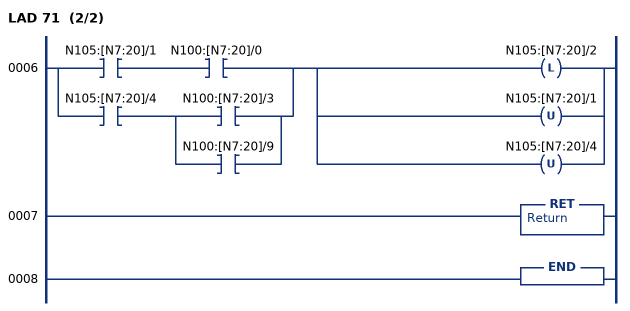
% Rung: 6 %
SOR BST XIC N105:[N7:20]/1 XIC N100:[N7:20]/0 NXB XIC N105:[N7:20]/4 BST XIC N100:[N7:20]/3 NXB XIC N100:[N7:20]/9 BND BND BST OTL N105:[N7:20]/2 NXB OTU N105:[N7:20]/1 NXB OTU N105:[N7:20]/4 BND EOR
% Rung: 7 %
SOR RET EOR
% Rung: 8 %
SOR END EOR

LADDER 75
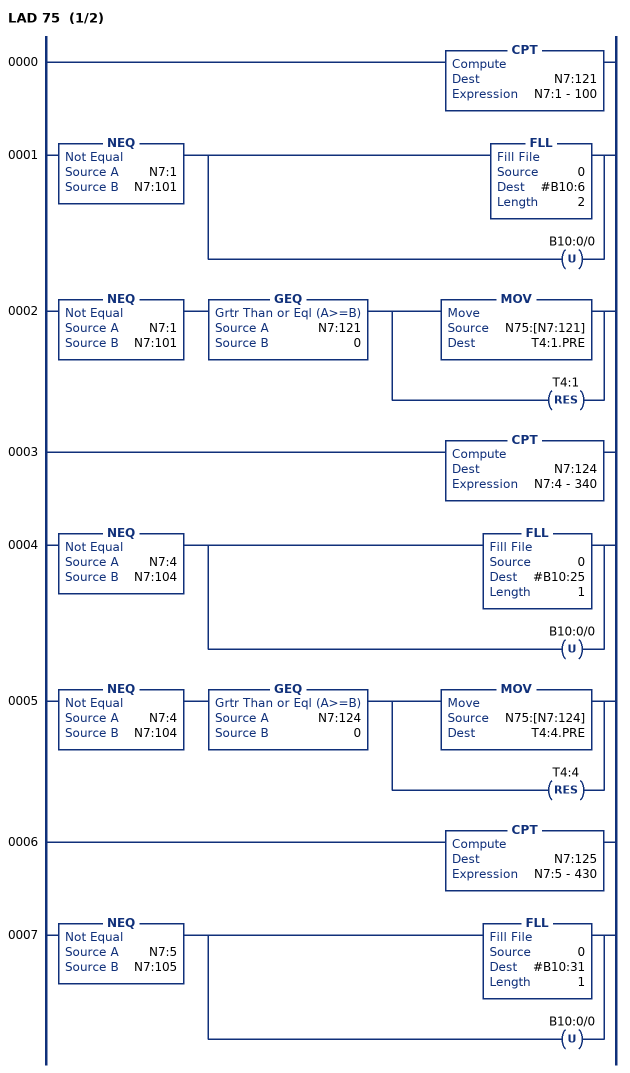
% Rung: 0 %
SOR CPT N7:121 " N7:1 - 100 " EOR
% Rung: 1 %
SOR NEQ N7:1 N7:101 BST FLL 0 #B10:6 2 NXB OTU B10:0/0 BND EOR
% Rung: 2 %
SOR NEQ N7:1 N7:101 GEQ N7:121 0 BST MOV N75:[N7:121] T4:1.PRE NXB RES T4:1 BND EOR
% Rung: 3 %
SOR CPT N7:124 " N7:4 - 340 " EOR
% Rung: 4 %
SOR NEQ N7:4 N7:104 BST FLL 0 #B10:25 1 NXB OTU B10:0/0 BND EOR
% Rung: 5 %
SOR NEQ N7:4 N7:104 GEQ N7:124 0 BST MOV N75:[N7:124] T4:4.PRE NXB RES T4:4 BND EOR
% Rung: 6 %
SOR CPT N7:125 " N7:5 - 430 " EOR
% Rung: 7 %
SOR NEQ N7:5 N7:105 BST FLL 0 #B10:31 1 NXB OTU B10:0/0 BND EOR

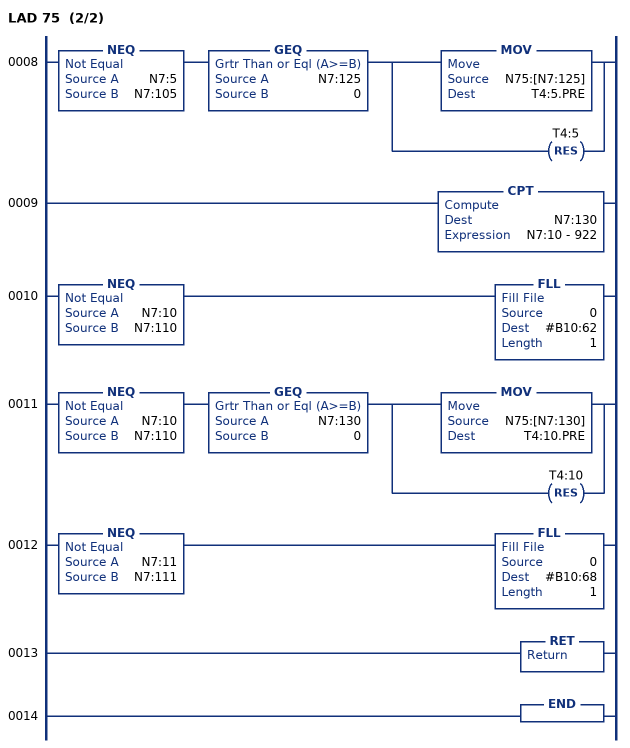
% Rung: 8 %
SOR NEQ N7:5 N7:105 GEQ N7:125 0 BST MOV N75:[N7:125] T4:5.PRE NXB RES T4:5 BND EOR
% Rung: 9 %
SOR CPT N7:130 " N7:10 - 922 " EOR
% Rung: 10 %
SOR NEQ N7:10 N7:110 FLL 0 #B10:62 1 EOR
% Rung: 11 %
SOR NEQ N7:10 N7:110 GEQ N7:130 0 BST MOV N75:[N7:130] T4:10.PRE NXB RES T4:10 BND EOR
% Rung: 12 %
SOR NEQ N7:11 N7:111 FLL 0 #B10:68 1 EOR
% Rung: 13 %
SOR RET EOR
% Rung: 14 %
SOR END EOR

LADDER 76
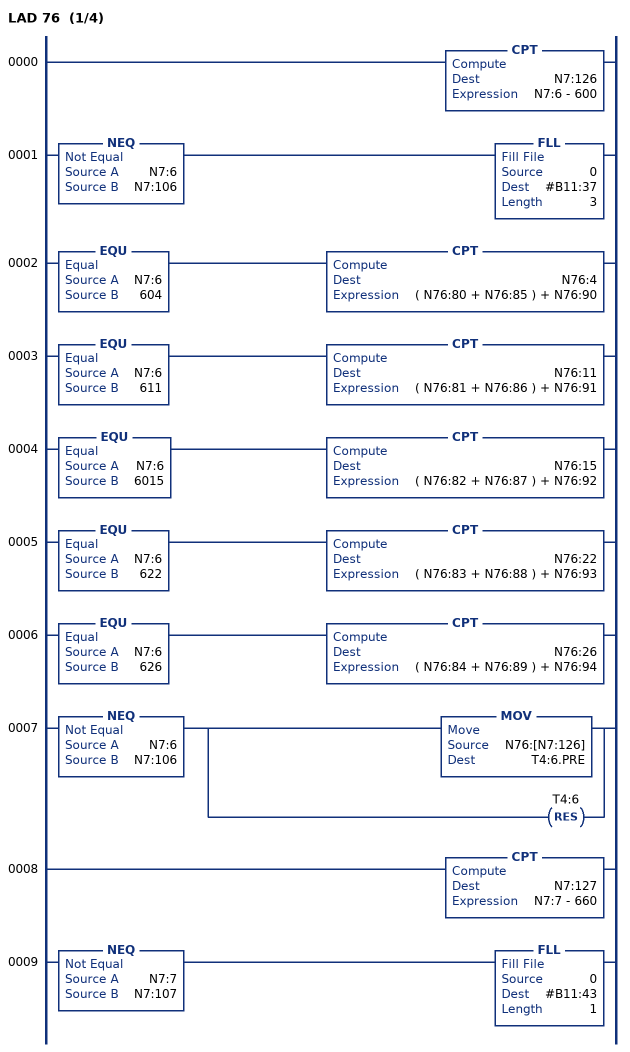
% Rung: 0 %
SOR CPT N7:126 " N7:6 - 600 " EOR
% Rung: 1 %
SOR NEQ N7:6 N7:106 FLL 0 #B11:37 3 EOR
% Rung: 2 %
SOR EQU N7:6 604 CPT N76:4 " ( N76:80 + N76:85 ) + N76:90 " EOR
% Rung: 3 %
SOR EQU N7:6 611 CPT N76:11 " ( N76:81 + N76:86 ) + N76:91 " EOR
% Rung: 4 %
SOR EQU N7:6 6015 CPT N76:15 " ( N76:82 + N76:87 ) + N76:92 " EOR
% Rung: 5 %
SOR EQU N7:6 622 CPT N76:22 " ( N76:83 + N76:88 ) + N76:93 " EOR
% Rung: 6 %
SOR EQU N7:6 626 CPT N76:26 " ( N76:84 + N76:89 ) + N76:94 " EOR
% Rung: 7 %
SOR NEQ N7:6 N7:106 BST MOV N76:[N7:126] T4:6.PRE NXB RES T4:6 BND EOR
% Rung: 8 %
SOR CPT N7:127 " N7:7 - 660 " EOR
% Rung: 9 %
SOR NEQ N7:7 N7:107 FLL 0 #B11:43 1 EOR

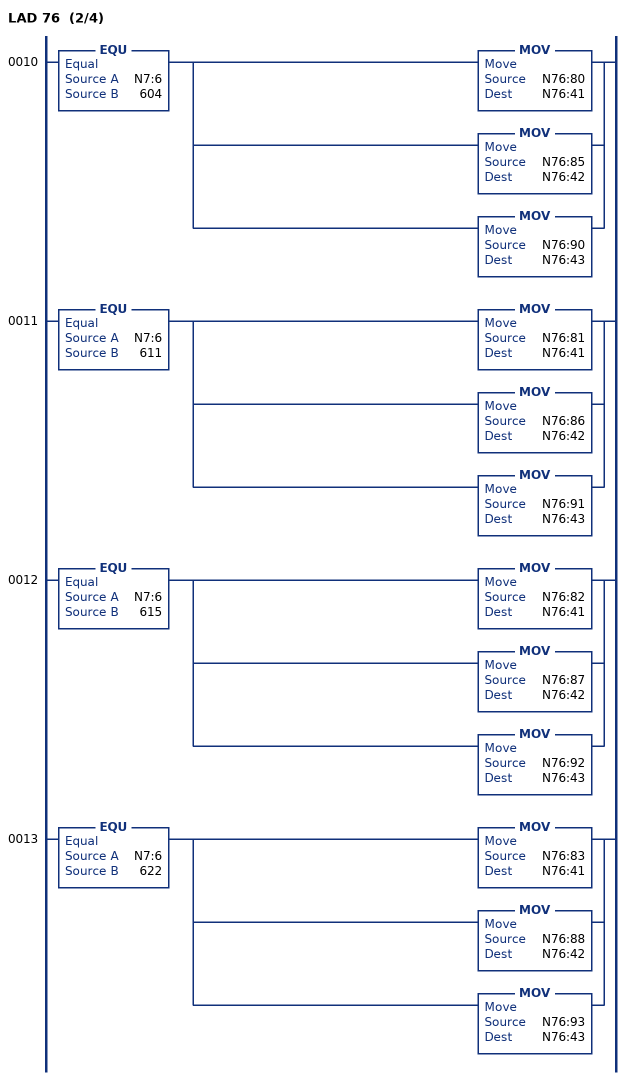
% Rung: 10 %
SOR EQU N7:6 604 BST MOV N76:80 N76:41 NXB MOV N76:85 N76:42 NXB MOV N76:90 N76:43 BND EOR
% Rung: 11 %
SOR EQU N7:6 611 BST MOV N76:81 N76:41 NXB MOV N76:86 N76:42 NXB MOV N76:91 N76:43 BND EOR
% Rung: 12 %
SOR EQU N7:6 615 BST MOV N76:82 N76:41 NXB MOV N76:87 N76:42 NXB MOV N76:92 N76:43 BND EOR
% Rung: 13 %
SOR EQU N7:6 622 BST MOV N76:83 N76:41 NXB MOV N76:88 N76:42 NXB MOV N76:93 N76:43 BND EOR

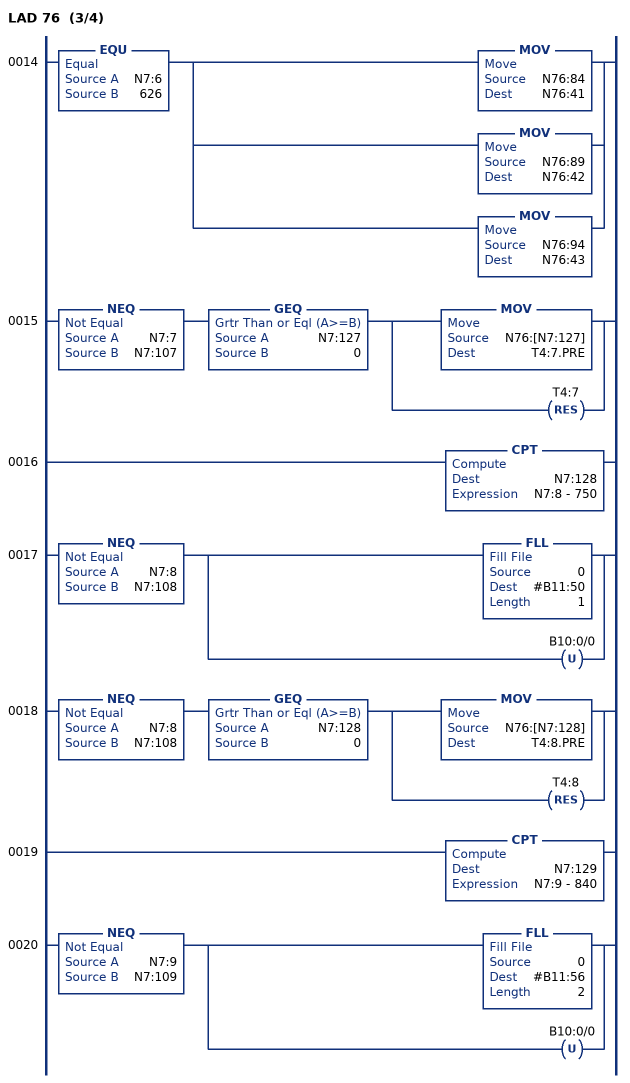
% Rung: 14 %
SOR EQU N7:6 626 BST MOV N76:84 N76:41 NXB MOV N76:89 N76:42 NXB MOV N76:94 N76:43 BND EOR
% Rung: 15 %
SOR NEQ N7:7 N7:107 GEQ N7:127 0 BST MOV N76:[N7:127] T4:7.PRE NXB RES T4:7 BND EOR
% Rung: 16 %
SOR CPT N7:128 " N7:8 - 750 " EOR
% Rung: 17 %
SOR NEQ N7:8 N7:108 BST FLL 0 #B11:50 1 NXB OTU B10:0/0 BND EOR
% Rung: 18 %
SOR NEQ N7:8 N7:108 GEQ N7:128 0 BST MOV N76:[N7:128] T4:8.PRE NXB RES T4:8 BND EOR
% Rung: 19 %
SOR CPT N7:129 " N7:9 - 840 " EOR
% Rung: 20 %
SOR NEQ N7:9 N7:109 BST FLL 0 #B11:56 2 NXB OTU B10:0/0 BND EOR

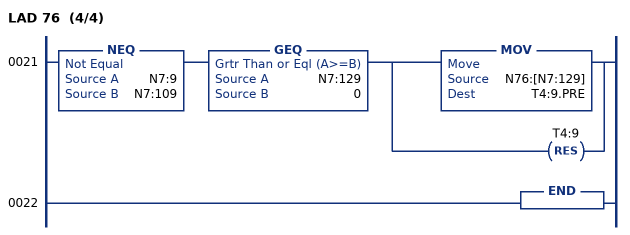
% Rung: 21 %
SOR NEQ N7:9 N7:109 GEQ N7:129 0 BST MOV N76:[N7:129] T4:9.PRE NXB RES T4:9 BND EOR
% Rung: 22 %
SOR END EOR

LADDER 77
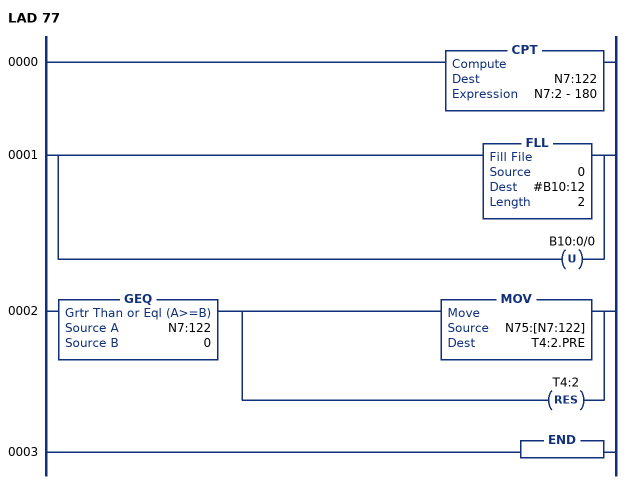
% Rung: 0 %
SOR CPT N7:122 " N7:2 - 180 " EOR
% Rung: 1 %
SOR BST FLL 0 #B10:12 2 NXB OTU B10:0/0 BND EOR
% Rung: 2 %
SOR GEQ N7:122 0 BST MOV N75:[N7:122] T4:2.PRE NXB RES T4:2 BND EOR
% Rung: 3 %
SOR END EOR

LADDER 78
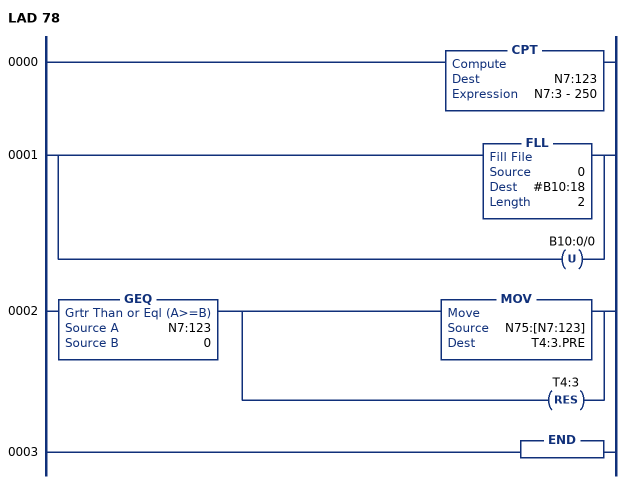
% Rung: 0 %
SOR CPT N7:123 " N7:3 - 250 " EOR
% Rung: 1 %
SOR BST FLL 0 #B10:18 2 NXB OTU B10:0/0 BND EOR
% Rung: 2 %
SOR GEQ N7:123 0 BST MOV N75:[N7:123] T4:3.PRE NXB RES T4:3 BND EOR
% Rung: 3 %
SOR END EOR

LADDER 80
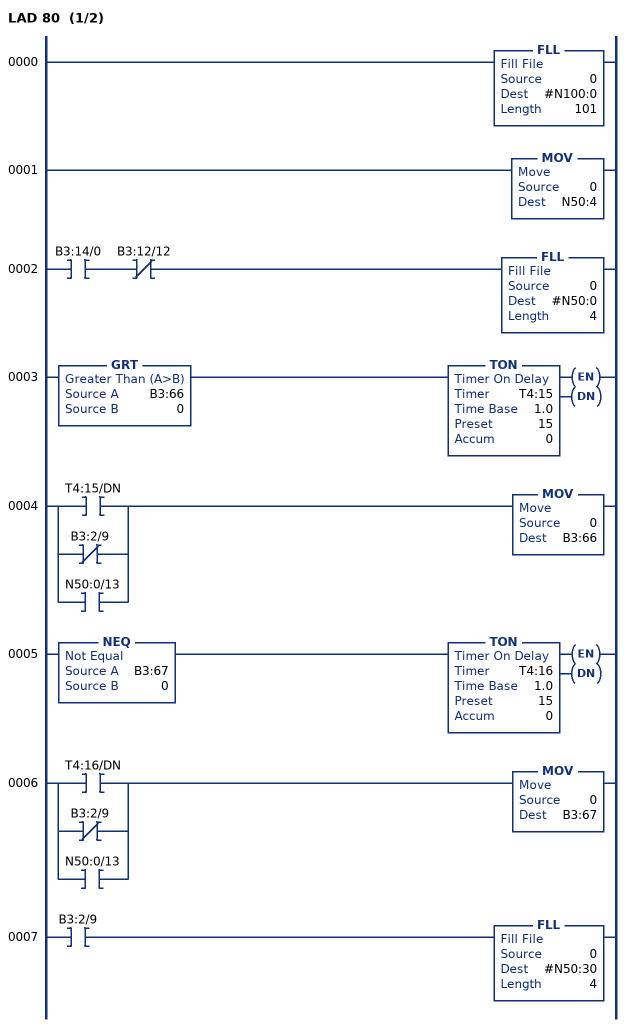
% Rung: 0 %
SOR FLL 0 #N100:0 101 EOR
% Rung: 1 %
SOR MOV 0 N50:4 EOR
% Rung: 2 %
SOR XIC B3:14/0 XIO B3:12/12 FLL 0 #N50:0 4 EOR
% Rung: 3 %
SOR GRT B3:66 0 TON T4:15 1.0 15 0 EOR
% Rung: 4 %
SOR BST XIC T4:15/DN NXB XIO B3:2/9 NXB XIC N50:0/13 BND MOV 0 B3:66 EOR
% Rung: 5 %
SOR NEQ B3:67 0 TON T4:16 1.0 15 0 EOR
% Rung: 6 %
SOR BST XIC T4:16/DN NXB XIO B3:2/9 NXB XIC N50:0/13 BND MOV 0 B3:67 EOR
% Rung: 7 %
SOR XIC B3:2/9 FLL 0 #N50:30 4 EOR

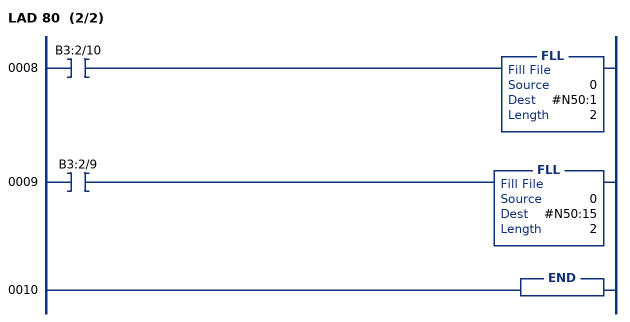
% Rung: 8 %
SOR XIC B3:2/10 FLL 0 #N50:1 2 EOR
% Rung: 9 %
SOR XIC B3:2/9 FLL 0 #N50:15 2 EOR
% Rung: 10 %
SOR END EOR

DATA TABLE (non-zero values as saved)
DATA B3
% B3:0 % 0X1006 0X6C09 0X0202 0X0000 0X0040 0X0000 0X0000 0X0100 0X0000 0X0800
% B3:10 % 0X0004 0X0000 0X0800 0X0000 0X0000 0X0000 0X0000 0X0000 0X0000 0X0000
% B3:20 % 0X0000 0X0000 0X0000 0X0000 0X0000 0X0400 0X0000 0X0000 0X0000 0X0000
% B3:60 % 0X0002 0X0001 0X0000 0X0000 0X8000 0X0000 0X0000 0X0000
DATA T4
% .PRE .ACC %
% T4:11 % 240 103
% T4:12 % 60 60
% T4:13 % 100 0
% T4:15 % 15 0
% T4:16 % 15 0
% T4:18 % 3600 0
% T4:19 % 32500 0
% T4:20 % 50 0
% T4:21 % 300 0
% T4:25 % 3600 0
% T4:26 % 600 0
% T4:28 % 200 0
% T4:30 % 50 47
% T4:31 % 50 0
DATA C5
% .PRE .ACC %
% C5:0 % 50 9
% C5:1 % 60 1
DATA R6
% .LEN .POS %
% R6:1 % 4 0
% R6:2 % 4 0
% R6:3 % 3 0
% R6:4 % 14 0
% R6:5 % 14 0
% R6:6 % 14 0
% R6:7 % 14 0
% R6:8 % 14 0
% R6:9 % 14 0
% R6:10 % 14 0
% R6:11 % 14 0
DATA N7
% N7:0 % 0 100 200 300 400 500 600 700 800 900
% N7:10 % 1000 1101 0 0 0 0 0 0 0 0
% N7:20 % 9 0 0 0 0 0 0 0 0 0
% N7:30 % 100 200 300 400 500 600 700 800 900 1000
% N7:40 % 1101 0 0 0 0 0 0 0 0 0
% N7:50 % 400 100 200 300 400 500 600 700 800 900
% N7:60 % 1000 200 200 0 0 0 0 0 0 0
% N7:80 % 1 0 0 0 0 0 0 0 0 0
% N7:100 % 0 100 200 300 400 500 600 700 800 900
% N7:110 % 1000 1101 0 0 0 0 0 0 0 0
% N7:120 % 0 0 20 50 60 70 0 40 50 60
% N7:130 % 78
DATA F8
% F8:5 % 0 0 0 43.33333 100
% F8:10 % 33.1333 0 0 0 0
DATA N9
% N9:0 % 10113 0 8192 0 0 0 0 0 0 0
% N9:10 % 2957 0 0 0 0 0 0 0 0 0
DATA B10
% B10:0 % 0X0000 0X0000 0X0000 0X0000 0X0000 0X0000 0X0010 0X0000 0X0000 0X0000
% B10:10 % 0X0000 0X0000 0X0100 0X0000 0X0000 0X0000 0X0000 0X0000 0X1000 0X0000
% B10:20 % 0X0000 0X0000 0X0000 0X0000 0X0000 0X0001 0X0000 0X0000 0X0000 0X0000
% B10:30 % 0X0000 0X0010 0X0000 0X0000 0X0000 0X0000 0X0000 0X0000 0X0000 0X0000
% B10:60 % 0X0000 0X0000 0X0100 0X0000 0X0000 0X0000 0X0000 0X0000 0X2000 0X0000
DATA B11
% B11:30 % 0X0000 0X0000 0X0000 0X0000 0X0000 0X0000 0X0000 0X0100 0X0000 0X0000
% B11:40 % 0X0000 0X0000 0X0000 0X1000 0X0000 0X0000 0X0000 0X0000 0X0000 0X0000
% B11:50 % 0X0001 0X0000 0X0000 0X0000 0X0000 0X0000 0X0010 0X0000 0X0000 0X0000
DATA T13
% .PRE .ACC %
% T13:0 % 300 0
% T13:1 % 120 0
DATA T21
% .PRE .ACC %
% T21:1 % 5 0
% T21:2 % 5 0
% T21:3 % 5 0
% T21:4 % 7 0
% T21:5 % 7 0
% T21:6 % 7 0
% T21:7 % 7 0
% T21:8 % 7 0
% T21:9 % 7 0
% T21:10 % 7 0
% T21:11 % 7 0
% T21:12 % 7 0
% T21:13 % 7 0
% T21:14 % 7 0
% T21:15 % 7 0
% T21:16 % 7 0
% T21:17 % 7 0
% T21:18 % 7 0
% T21:19 % 5 5
% T21:20 % 5 0
% T21:21 % 5 5
% T21:22 % 5 5
% T21:23 % 5 5
% T21:24 % 5 5
% T21:25 % 5 0
% T21:26 % 5 0
% T21:27 % 15 0
% T21:28 % 7 0
% T21:29 % 5 5
% T21:30 % 5 5
% T21:31 % 5 5
% T21:32 % 5 0
% T21:33 % 5 0
% T21:34 % 5 5
% T21:35 % 5 0
% T21:37 % 300 0
% T21:38 % 5 0
% T21:39 % 5 5
% T21:40 % 5 0
% T21:41 % 5 0
% T21:42 % 5 5
% T21:43 % 30 0
% T21:44 % 70 0
% T21:45 % 1 0
% T21:46 % 20 0
% T21:47 % 30 0
% T21:48 % 5 5
% T21:49 % 10 0
% T21:50 % 10 0
% T21:51 % 120 0
% T21:52 % 120 0
% T21:53 % 120 0
% T21:54 % 120 0
% T21:55 % 120 0
% T21:56 % 120 0
% T21:57 % 120 0
% T21:58 % 120 0
% T21:59 % 15 0
% T21:60 % 15 0
% T21:61 % 5 0
% T21:62 % 120 0
% T21:63 % 30 0
% T21:64 % 1 0
DATA B22
% B22:0 % 0X0000 0X0000 0X0000 0X0000 0X0000 0X0780 0X0000 0X0000 0X313C 0X0000
DATA N25
% N25:10 % 0 9 0 0 0 0 0 0 0 0
% N25:20 % 0 50 20 100 50 100 130 20 0 0
% N25:30 % 0 1256 1150 1000 1150 1100 650 0 0 0
% N25:40 % 0 1240 1150 1100 1150 0 0 0 0 0
% N25:50 % 0 289 1050 1050 0 0 0 0 0 0
% N25:60 % 0 11196 1000 20 120 60 373 30000 373 0
% N25:80 % 0 0 100 100 0 0 0 0 0 0
% N25:90 % 0 1172 1100 1250 1100 0 0 0 44 100
% N25:100 % 0 0 1100 1250 1100 0 0 0 0 0
% N25:110 % 0 0 1380 0 1380 0 0 0 0 0
% N25:120 % 0 0 0 1100 1250 0 0 0 0 0
% N25:130 % 0 0 0 1100 650 0 0 0 0 0
% N25:140 % 0 0 0 650 0 0 0 0 0 0
% N25:160 % 0 0 0 0 1262 0 0 2500 2200 0
% N25:170 % 0 289 0 2500 2200 0 0 0 0 0
% N25:180 % 0 0 0 2500 0 0 0 0 0 0
% N25:190 % 0 0 0 2500 0 0 0 0 0 0
DATA B29
% B29:0 % 0X0200 0X0000 0X0000 0X0000 0X0000 0X0000 0X0000 0X0000 0X0000 0X0000
DATA T31
% .PRE .ACC %
% T31:0 % 5 0
% T31:1 % 60 0
% T31:2 % 300 0
% T31:3 % 4 0
% T31:4 % 300 12
% T31:5 % 4 0
% T31:6 % 5 0
% T31:7 % 60 0
% T31:8 % 10 0
% T31:9 % 10 0
% T31:10 % 10 0
% T31:11 % 15 0
% T31:12 % 10 0
% T31:13 % 5 0
% T31:14 % 10 0
% T31:15 % 7 0
% T31:16 % 60 0
% T31:17 % 40 0
% T31:18 % 5 0
% T31:19 % 60 0
% T31:20 % 5 0
% T31:21 % 3 0
% T31:22 % 1800 0
% T31:23 % 1800 0
% T31:24 % 600 0
% T31:25 % 600 0
% T31:26 % 60 0
% T31:27 % 60 0
% T31:28 % 15 0
% T31:29 % 15 0
% T31:30 % 60 0
% T31:31 % 5 0
% T31:32 % 3600 0
% T31:33 % 7 0
% T31:34 % 15 0
% T31:35 % 15 0
% T31:36 % 10 9
% T31:37 % 10 0
% T31:38 % 300 0
% T31:39 % 1 0
DATA N32
% N32:0 % 0 12000 0 0 0 0 0 2957 0 0
% N32:10 % 0 6242 6242 0
DATA N40
% N40:0 % -24555 0 7645 100 8 0 0 16383 0 0
% N40:10 % 0 100 0 4 7602 -43 42 6847 -30648 1
% N40:20 % -9440 6487 7645 7602 6804 0 0 260 120 140
% N40:30 % 145 0 100 0 0 0 0 0 0 0
% N40:40 % 0 240 60 140 139 415 415 5 0 100
% N40:50 % 0 0 5 0 0 0 0 0 13608 0
DATA N41
% N41:0 % 17 4352 8192 100 8 0 0 16383 0 0
% N41:10 % 0 100 0 4 0 -8192 0 0 0 0
% N41:20 % 0 313 8192 0 0 0 0 800 800 0
% N41:40 % 0 0 0 800 0 0 0 5 0 100
% N41:50 % 0 0 5 0 0 0 0 0 0 0
DATA N42
% N42:10 % 0 100 0 0 0 0 0 0 0 0
% N42:60 % 0 0 0 0 0 0 0 16383 0 0
DATA B49
% B49:0 % 0X0008 0X0000
DATA N50
% N50:50 % 9 1 0 0
DATA N51
% N51:0 % 0 0 16388 -6592 2 0 0 0 0 0
% N51:10 % 0 0 0 0 0 0 0 1 1 0
% N51:50 % 0 16 80 0 2 0 0 0 0 0
% N51:60 % 1 32 1 21 0 81 64 0 64 64
% N51:70 % 64 34 0 0 0 0 0 0 2 0
% N51:90 % 0 0 0 0 0 0 700 0 900 0
% N51:100 % 1101 0 200 0 300 0 400 0 800 0
% N51:110 % 400 0 0 0 0 0 0 0 0 3
% N51:120 % 0 0 0 0 0 0 0 0 0 10
% N51:130 % 1 5 1 1 5 5 6 0 1239 1239
% N51:140 % 289 0 373 139 1239 1239 289 0 373 139
% N51:150 % 44 0 0 0 0 0 0 0 0 0
% N51:200 % 127 1 1 1 1 1 1 1 1 0
DATA B53
% B53:0 % 0X0002 0X0000 0X0000 0X0000 0X0000 0X0000 0X0000 0X0000 0X0000 0X0000
% B53:10 % 0X0000 0X0000 0X0000 0X0000 0X0000 0X0000 0X3030 0X0055 0X6404 0X400A
DATA N54
% N54:0 % -32602 160 0 0 0 0 0 0 0 0
% N54:10 % 8192 0 0 0 0 0 0 0 0 0
% N54:20 % -32512 0 0 0 0 0 0 0 0 0
% N54:30 % -32768
DATA N60
% N60:0 % -31744 2 1 54 137 10 0 228 5 5
% N60:10 % 0 2 256 0 0 0 0 0 0 0
% N60:20 % -24576 3 1 231 137 46 0 224 5 4
% N60:30 % 0 2 3072 0 0 0 0 0 0 0
% N60:40 % -24576 3 1 231 137 6 0 160 5 4
% N60:50 % 0 2 3072 0
DATA N75
% N75:0 % 0 30 10 5 120 5 60 5 0 0
% N75:10 % 30 0 1800 300 750 85 20 0 0 0
% N75:20 % 0 60 10 10 5 2 2 0 0 0
% N75:30 % 2 5 5 5 5 10 10 15 0 0
% N75:40 % 10 0 0 0 0 0 0 0 0 0
% N75:50 % 0 2 3 0 3 10 0 0 0 0
% N75:60 % 0 0 600 0 650 0 0 0 0 0
% N75:70 % 0 0 300 0 0 0 0 0 0 0
% N75:80 % 0 90 52 16 50 70 35 70 55 0
% N75:240 % 70 70 35 70 55 0 0 0 0 0
DATA N76
% N76:0 % 0 0 5 300 50 60 5 30 0 0
% N76:10 % 1800 65 1800 5 300 55 60 5 0 0
% N76:20 % 30 600 55 120 5 360 50 180 0 0
% N76:30 % 5 0 120 0 0 0 0 0 0 0
% N76:40 % 0 30 15 5 0 0 0 0 0 0
% N76:50 % 0 0 0 15 10 0 0 0 0 0
% N76:60 % 0 300 60 1200 30 300 60 600 0 0
% N76:70 % 30 300 300 0 0 0 0 0 0 0
% N76:80 % 30 30 30 30 30 15 30 20 20 15
% N76:90 % 5 5 5 5 5 0 0 0 0 0
DATA N90
% N90:0 % 112 1800 1800 0 112
DATA N91
% N91:0 % 0 30 10 5 120 5 60 5 0 0
% N91:10 % 30 0 1800 300 750 85 20 0 0 0
% N91:20 % 0 60 10 10 5 2 2 0 0 0
% N91:30 % 2 5 5 5 5 10 10 15 0 0
% N91:40 % 10 0 0 0 0 0 0 0 0 0
% N91:50 % 0 2 3 0 3 10 0 0 0 0
% N91:60 % 0 0 600 0 650 0 0 0 0 0
% N91:70 % 0 0 300 0 0 0 0 0 0 0
% N91:80 % 0 90 52 16 50 70 35 70 55 0
% N91:100 % 0 0 5 300 50 60 5 30 0 0
% N91:110 % 1800 65 1800 5 300 55 60 5 0 0
% N91:120 % 30 600 55 120 5 360 50 180 0 0
% N91:130 % 5 0 120 0 0 0 0 0 0 0
% N91:140 % 0 30 15 5 0 0 0 0 0 0
% N91:150 % 0 0 0 15 10 0 0 0 0 0
% N91:160 % 0 300 60 1200 30 300 60 600 0 0
% N91:170 % 30 300 300 0 0 0 0 0 0 0
% N91:180 % 30 30 30 30 30 15 30 20 20 15
% N91:190 % 5 5 5 5 5 0 0 0 0 0
% N91:220 % 5 0 0 0 1600 1590 300 0 0 0
% N91:240 % 97 0 0 0 0 0 0 0 0 1
DATA N92
% N92:0 % 50 20 100 20 100 130 1250 1100 650 650
% N92:10 % 1250 1100 1250 950 100 150 120 0 12000 0
% N92:20 % 0 0 0 0 0 100 1250 1100 1250 1100
% N92:30 % 0 1380 1100 1250 1100 650 650 0 0 0
% N92:40 % 0 1262 0 0 0 0 0 0 0 0
DATA N105
% N105:0 % 0 -32767 2 2 -32767 2 -32767 -32767 -32767 -32767
